PROGRAM Z_Axis
VAR
	HMI_Z_UP : BOOL;
	HMI_Z_DOWN : BOOL;
END_VAR

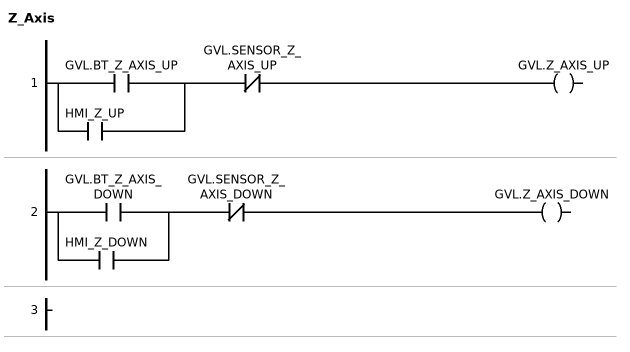
// NETWORK 1
GVL.Z_AXIS_UP := (GVL.BT_Z_AXIS_UP OR HMI_Z_UP) AND NOT GVL.SENSOR_Z_AXIS_UP;

// NETWORK 2
GVL.Z_AXIS_DOWN := (GVL.BT_Z_AXIS_DOWN OR HMI_Z_DOWN) AND NOT GVL.SENSOR_Z_AXIS_DOWN;

// NETWORK 3

END_PROGRAM

(* stored: Version 1.1.0.1, ProductVersion 3.1.4024.13
   POU Z_Axis: Id {52882fe4-2fda-499c-8884-f8d524738b5b}, SpecialFunc None *)
